FUNCTION_BLOCK FB_MyLocalObjectEvents EXTENDS FB_BA_LocalObjectEventSubscriber

METHOD PRIVATE IsPressure : BOOL
VAR_INPUT
	eUnit		: E_BA_Unit;
END_VAR
IsPressure := (E_BA_Unit.ePressure_Pascals <= eUnit) AND_THEN (eUnit <= E_BA_Unit.ePressure_InchesOfMercury);
END_METHOD

METHOD PRIVATE IsTemperature : BOOL
VAR_INPUT
	eUnit		: E_BA_Unit;
END_VAR
IsTemperature := (E_BA_Unit.eTemperature_DegreesCelsius <= eUnit) AND_THEN (eUnit <= E_BA_Unit.eTemperature_DegreeDaysFahrenheit);
END_METHOD

METHOD PROTECTED OnInitInstanceId
VAR_INPUT
	iObject			: I_BA_Object;
END_VAR
VAR_INST
	_nID_Temp		: UDINT						:= 5000;				// First ID to assign to temperature sensors.
	_nID_Prs		: UDINT						:= 6000;				// First ID to assign to pressure sensors.
END_VAR
VAR
	_iAnalogObj		: I_BA_AnalogObject;
	_nID			: REFERENCE TO UDINT;
END_VAR
// Sample 1) Generate instance ID related to configured units.

IF (iObject.InstanceID <> 0) THEN
	; // ID already assigned.
ELSIF (iObject.DataClass <> E_BA_DataClass.eAnalog) THEN
	; // Skip.
ELSIF (NOT __QUERYINTERFACE(iObject, _iAnalogObj)) THEN
	; // Failed to convert interface.
ELSE
	// Determine range of instance IDs:
	IF (IsTemperature(_iAnalogObj.Unit)) THEN
		_nID REF= _nID_Temp;
	ELSIF (IsPressure(_iAnalogObj.Unit)) THEN
		_nID REF= _nID_Prs;
	ELSE
		RETURN; // Skip (Instance ID will be auto-generated).
	END_IF
		
	// Assign instance ID:
	_iAnalogObj.InstanceID := _nID;
	iObject.LogMsg.Show1(ADSLOG_MSGTYPE_HINT, 'OIII21', 'Assigned instance ID %d.', F_UDINT(_nID), FALSE);
	
	_nID := (_nID+1);
END_IF
END_METHOD

END_FUNCTION_BLOCK

(* stored: Version 1.1.0.1, ProductVersion 3.1.4024.9
   POU FB_MyLocalObjectEvents: Id {435807dc-5aae-4d12-89bc-d25a17ff58e3}, SpecialFunc None
   Folder [Private] Helper: Id {9d9a0465-d4d4-48d9-9c35-4f244b497295}
   Folder [Protected] Events: Id {cca82e83-5f4b-4811-b7c2-04e15e3ebc6d}
   Method IsPressure: Id {5aaf513d-5ef4-4794-b1ab-187dfd790870}
   Method IsTemperature: Id {9cf25a15-9b02-43f6-9b1c-924566998260}
   Method OnInitInstanceId: Id {c9f9993e-e237-4917-8299-2a47d61c3632} *)
